FUNCTION_BLOCK SEM (* Basic Function Block Type *)
  (* Standard: 61499-2 *)
  (* Version 0.3, 2009-09-15, JHC, Holobloc Inc, Changed transition priorities. *)
  (* Version 0.2, 2003-12-04, JHC, Rockwell Automation, Renamed for better indexing. *)
  (* Version 0.1, 2002-11-05, JHC, Rockwell Automation, Corrected missing ST element in Algorithm REQ. *)
  (* Version 0.0, 2000-05-30, JHC, Rockwell Automation *)
  PACKAGE fb.rt.DIAS;
  IMPORT fb.datatype.*;
  IMPORT fb.rt.*;
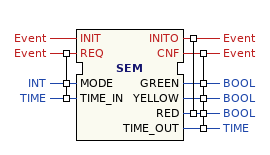
  EVENT_INPUT
    INIT; (* Initialization Request *)
    REQ WITH MODE, TIME_IN;
  END_EVENT
  EVENT_OUTPUT
    INITO WITH RED; (* Initialization Confirm *)
    CNF WITH GREEN, YELLOW, RED, TIME_OUT;
  END_EVENT
  VAR_INPUT
    MODE : INT;
    TIME_IN : TIME;
  END_VAR
  VAR_OUTPUT
    GREEN : BOOL;
    YELLOW : BOOL;
    RED : BOOL;
    TIME_OUT : TIME;
  END_VAR
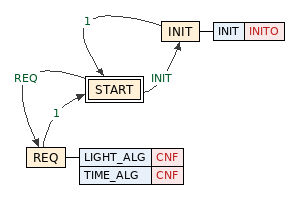
  EC_STATES
    START; (* Initial State *)
    INIT : INIT -> INITO; (* Initialization *)
    REQ : LIGHT_ALG -> CNF, TIME_ALG -> CNF;
  END_STATES
  EC_TRANSITIONS
    INIT TO START := 1;
    START TO INIT := INIT;
    START TO REQ := REQ;
    REQ TO START := 1;
  END_TRANSITIONS
  ALGORITHM INIT IN ST: (* Initialization algorithm *)
GREEN := false;
YELLOW := false;
RED := true;
  END_ALGORITHM
  ALGORITHM LIGHT_ALG IN ST:
IF MODE = 0 THEN
	GREEN := false;
	YELLOW := false;
	RED := true;
END_IF

IF MODE = 1 THEN
	GREEN := false;
	YELLOW := true;
	RED := false;
END_IF

IF MODE = 2 THEN
	GREEN := true;
	YELLOW := false;
	RED := false;
END_IF
  END_ALGORITHM
  ALGORITHM TIME_ALG IN ST:
TIME_OUT := TIME_IN;
  END_ALGORITHM
END_FUNCTION_BLOCK
